Universal Robots PolyScope program: test1.urp

Program test1 (installation=default directory=/programs createdIn=3.10.1.76190 lastSavedIn=3.10.1.76190 robotSerialNumber=2017356443)
Calibrated DH parameters: a=[0.000092, -0.116521, -0.182101, -0.000106, 0.000044, 0]; d=[0.089391, 255.189113, -82.629387, -172.449369, 0.094782, 0.082637]; alpha=[1.569598, 0.001603, 0.002015, 1.570234, -1.570307, 0]; deltaTheta=[-0.000017, 1.293309, -0.204843, -1.088417, 0.000036, -0.000078]
Robot Program (runOnlyOnce=false)
  MoveJ speed 60 deg/s, acceleration 80 deg/s^2 (useActiveTCP=true)
    Waypoint Waypoint_1: TCP in base x=391.308 y=-192.864 z=800.596 mm, rx=0.0256 ry=-2.2092 rz=2.2084 rad; joints [0.106, -92.132, -57.397, -53.584, -0.023, 21.729] deg
    Waypoint Waypoint_2 (Variable): variable(featureName=bucket)
